FUNCTION_BLOCK ControllerCentralised (* Basic Function Block Type *)
  (* Standard: 61499-2 *)
  (* Version 0.3, 2009-09-15, JHC, Holobloc Inc, Changed transition priorities. *)
  (* Version 0.2, 2003-12-04, JHC, Rockwell Automation, Renamed for better indexing. *)
  (* Version 0.1, 2002-11-05, JHC, Rockwell Automation, Corrected missing ST element in Algorithm REQ. *)
  (* Version 0.0, 2000-05-30, JHC, Rockwell Automation *)
  (* Compiler header: package fb.rt.template; *)
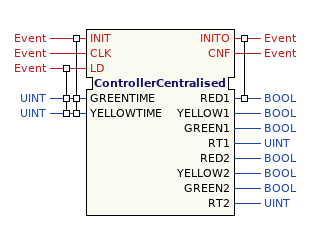
  EVENT_INPUT
    INIT WITH GREENTIME, YELLOWTIME; (* Initialization Request *)
    CLK; (* Normal Execution Request *)
    LD WITH GREENTIME, YELLOWTIME;
  END_EVENT
  EVENT_OUTPUT
    INITO WITH RED1; (* Initialization Confirm *)
    CNF;
  END_EVENT
  VAR_INPUT
    GREENTIME : UINT;
    YELLOWTIME : UINT;
  END_VAR
  VAR_OUTPUT
    RED1 : BOOL; (* Output event qualifier *)
    YELLOW1 : BOOL;
    GREEN1 : BOOL;
    RT1 : UINT;
    RED2 : BOOL;
    YELLOW2 : BOOL;
    GREEN2 : BOOL;
    RT2 : UINT;
  END_VAR
  VAR
    RELEASE : BOOL;
    GREENTIME1CV : UINT;
    GREENTIME2CV : UINT;
    YELLOWTIME1CV : UINT;
    YELLOWTIME2CV : UINT;
  END_VAR
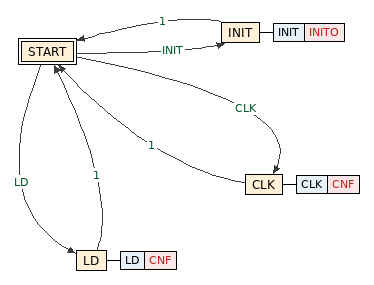
  EC_STATES
    START; (* Initial State *)
    INIT : INIT -> INITO; (* Initialization *)
    CLK : CLK -> CNF; (* Normal execution *)
    LD : LD -> CNF;
  END_STATES
  EC_TRANSITIONS
    INIT TO START := 1;
    START TO CLK := CLK;
    START TO INIT := INIT;
    CLK TO START := 1;
    START TO LD := LD;
    LD TO START := 1;
  END_TRANSITIONS
  ALGORITHM INIT IN ST: (* Initialization algorithm *)
RED1:=FALSE;
YELLOW1:=FALSE;
GREEN1:=FALSE;
RED2:=FALSE;
YELLOW2:=FALSE;
GREEN2:=FALSE;
RELEASE:=FALSE;
  END_ALGORITHM
  ALGORITHM CLK IN ST: (* Normally executed algorithm *)
IF RELEASE = FALSE THEN
	IF GREENTIME1CV > 0 THEN
		GREENTIME1CV := GREENTIME1CV - 1;
		GREEN1:=TRUE;
		YELLOW1:= FALSE;
		RED1:=FALSE;
		GREEN2:=FALSE;
		YELLOW2:= FALSE;
		RED2:=TRUE;
		RT1:=GREENTIME1CV;
	END_IF;

	IF  GREENTIME1CV=0 THEN
		GREEN1:=FALSE;
		YELLOW1:= TRUE;
		RED1:=FALSE;
		GREEN2:=FALSE;
		YELLOW2:= FALSE;
		RED2:=TRUE;
		IF YELLOWTIME1CV>0 THEN
			YELLOWTIME1CV:= YELLOWTIME1CV - 1;
			RT1:=YELLOWTIME1CV;
		END_IF;
	END_IF;
	IF YELLOWTIME1CV=0 THEN
		GREEN1:=FALSE;
		YELLOW1:=FALSE;
		RED1:=TRUE;
		GREEN2:=TRUE;
		YELLOW2:=FALSE;
		RED2:=FALSE;
		RELEASE:=TRUE;
		RT1:=0;
		RT2:=GREENTIME;
		GREENTIME1CV:= GREENTIME;
		YELLOWTIME1CV:=  YELLOWTIME;
	END_IF;
END_IF;

IF RELEASE = TRUE THEN
	IF GREENTIME2CV > 0 THEN
		GREENTIME2CV := GREENTIME2CV - 1;
		GREEN1:=FALSE;
		YELLOW1:= FALSE;
		RED1:=TRUE;
		GREEN2:=TRUE;
		YELLOW2:= FALSE;
		RED2:=FALSE;
		RT1:=0;
		RT2:=GREENTIME2CV;
	END_IF;
	IF GREENTIME2CV=0 THEN
		GREEN1:=FALSE;
		YELLOW1:= FALSE;
		GREEN2:=FALSE;
		YELLOW2:= TRUE;
		RED2:=FALSE;
		IF YELLOWTIME2CV>0 THEN
			YELLOWTIME2CV:= YELLOWTIME2CV - 1;
		    RT2:=YELLOWTIME2CV;
		END_IF;
	END_IF;
	IF YELLOWTIME2CV=0 THEN
		GREEN1:=TRUE;
		YELLOW1:=FALSE;
		RED1:=FALSE;
		GREEN2:=FALSE;
		YELLOW2:=FALSE;
		RED2:=TRUE;
		RELEASE:=FALSE;
		RT1:=GREENTIME;
		RT2:=0;
		GREENTIME2CV:= GREENTIME;
		YELLOWTIME2CV:=  YELLOWTIME;
	END_IF;
END_IF;
  END_ALGORITHM
  ALGORITHM LD IN ST:
GREEN1:=TRUE;
YELLOW1:=FALSE;
RED1:=FALSE;
GREEN2:=FALSE;
YELLOW2:=FALSE;
RED2:=TRUE;

RT1:=GREENTIME;
RT2:= 0;
GREENTIME1CV:=GREENTIME;
GREENTIME2CV:=GREENTIME;
YELLOWTIME1CV:=YELLOWTIME+1;
YELLOWTIME2CV:=YELLOWTIME+1;
  END_ALGORITHM
END_FUNCTION_BLOCK
